{attribute 'qualified_only'}
{attribute 'strict'}
TYPE E_REGIO_SELECTION :
(
	USA := 0,
	EUROPE
);
END_TYPE

(* stored: Version 1.1.0.1, ProductVersion 3.1.4026.18
   DUT E_REGIO_SELECTION: Id {e878dd7d-1541-4518-a44c-9361162d8dda} *)
